(* PLC project Unnamed, Unknown Unnamed 1 *)
(* stored: creationDateTime 2021-01-21T10:01:36, modificationDateTime 2021-01-22T21:40:23 *)

PROGRAM program1
  VAR
    PB1 AT %IX100.0 : BOOL;
    PB2 AT %IX100.1 : BOOL;
    LAMP AT %QX100.0 : BOOL;
  END_VAR

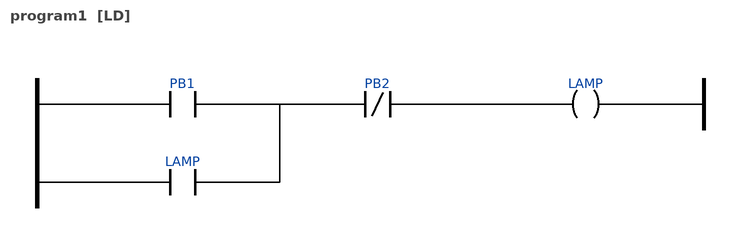
(* LD diagram, written out as Structured Text *)
LAMP := (PB1 OR LAMP) AND NOT PB2;
END_PROGRAM

CONFIGURATION Config0
  RESOURCE Res0 ON PLC
    TASK task0(INTERVAL := T#20ms, PRIORITY := 0);
    PROGRAM instance0 WITH task0 : program1;
  END_RESOURCE
END_CONFIGURATION
